{attribute 'GeneratedUsingTerminal: AT2041-0250-0022'}
{attribute addProperty BoxType "AT2041-0250-0022"}
{attribute addProperty Id "A_0100_AT2040_5250_0019_AT2040_5250AT2040_01D6DEDF80"}
{attribute addProperty CRC "3355827542"}
{attribute addProperty Size "80"}
TYPE A_0044_AT2041_0250_0022_C805DD56 EXTENDS AT2041_86175B41 :
STRUCT
	{attribute addProperty Name "A_0100_AT2040_5250_0019_AT2040_5250"}
	{attribute addProperty PreviousPort "A_0044(AT2041-0250-0022) : B"}
	A_0100_AT2040_5250_0019_AT2040_5250 : AT2040_01D6DEDF;
END_STRUCT
END_TYPE

(* stored: Version 1.2.0.0, ProductVersion 3.1.4024.9
   DUT A_0044_AT2041_0250_0022_C805DD56: Id {b4f92dbc-a035-4fc3-a91f-204c383ce3e7} *)
